// TIA Portal V15.1 export
// export: Created 2024-05-17T05:38:54.2339682Z, ExportSetting WithDefaults, DisplayName Totally Integrated Automation Portal, DisplayVersion V15.1 Update 5, DisplayName TIA Portal Openness, DisplayVersion V15.1 Update 5, DisplayName SINAMICS Startdrive Advanced, DisplayVersion V15.1, DisplayName G130, G150, S120, S150, SINAMICS MV, S210, DisplayVersion V15.1, DisplayName G110M, G120, G120C, G120D, G120P, DisplayVersion V15.1, DisplayName STEP 7 Professional, DisplayVersion V15.1 Update 5, DisplayName STEP 7 Safety, DisplayVersion V15.1, DisplayName WinCC Professional, DisplayVersion V15.1 Update 5, DisplayName SIMATIC Visualization Architect, DisplayVersion V15.1
FUNCTION_BLOCK "LAndonReqVCG"   // FB6050, FBD
TITLE = FB6050: LandonReq / FB6050: LandonReq VCG
{ S7_Optimized_Access := 'FALSE' }
VERSION : 0.1
// =============================================================================
// This module:
//  * Evaluate the Pullcord request to trigger an ANDON event
//  * Gather and organise the data to send to IT shopfloor
//  * Send data to Andon Server on change (buffers only when changed and after 30 
//    sec without an active send)
// =============================================================================
// 08/06/2017: Added Lmaintenancesel
//                       changed Send done to local varible
// 14/02/2017: APPROVAL TEST WITH IT
// 07/12/2106: Expanded StationId to 14 characters
// ============================================================================
// This module:25/11/2016
//  * Evaluate the HCall request to trigger an ANDON event
//  * Gather and organise the data to send to IT shopfloor
//  * Send data to Andon Server on change (buffers only when changed and after 30 
//    sec without an active send)
// ============================================================================
// stored: AutoNumber false, IsIECCheckEnabled false, SetENOAutomatically False, UDAEnableTagReadback false
   VAR_INPUT
      I_WaitingInput { ExternalAccessible := 'False'; ExternalVisible := 'False'; ExternalWritable := 'False'} : Bool;   // I: Not enough bodies on input
      I_WaitingOutput { ExternalAccessible := 'False'; ExternalVisible := 'False'; ExternalWritable := 'False'} : Bool;   // I: Can't deliver body on output
      I_LineStop { ExternalAccessible := 'False'; ExternalVisible := 'False'; ExternalWritable := 'False'} : Bool;   // I: Line Stop
      I_AutoZoneOverCycle { ExternalAccessible := 'False'; ExternalVisible := 'False'; ExternalWritable := 'False'} : Bool;   // I: Automatic unit has exceeded reference time
      I_Operator1OverCycle { ExternalAccessible := 'False'; ExternalVisible := 'False'; ExternalWritable := 'False'} : Bool;   // I: Operator has exceeded reference time
      I_Operator2OverCycle { ExternalAccessible := 'False'; ExternalVisible := 'False'; ExternalWritable := 'False'} : Bool;   // I: Operator has exceeded reference time
      I_Operator3OverCycle { ExternalAccessible := 'False'; ExternalVisible := 'False'; ExternalWritable := 'False'} : Bool;   // I: Operator has exceeded reference time
      I_Operator4OverCycle { ExternalAccessible := 'False'; ExternalVisible := 'False'; ExternalWritable := 'False'} : Bool;   // I: Operator has exceeded reference time
      I_Operator5OverCycle { ExternalAccessible := 'False'; ExternalVisible := 'False'; ExternalWritable := 'False'} : Bool;   // I: Operator has exceeded reference time
      I_Mask { ExternalAccessible := 'False'; ExternalVisible := 'False'; ExternalWritable := 'False'} : Bool;   // I: Mask Andon
   END_VAR
   VAR_IN_OUT
      IO_Modes : "Modes";   // IO: Modes
      IO_VD : "VDComm";   // IO: VDCOM
      IO_AndonStatusVCG : "AndonStatusVCG";   // IO: AndonStatus / IO: AndonStatus <-> Supervision
      IO_AndonDataExchange : "AndonDataExchangeVCG";   // IO: AndonDataExchange
      H_HMI : "H_HMI";   // IO: HMO
      H_AndonReq : "H_AndonReqVCG";   // IO: H_Andon Req
      C_Config : "AndonConfigVCG";   // IO: AndonConfig
   END_VAR
   VAR DB_SPECIFIC
      HCall0 { ExternalAccessible := 'False'; ExternalVisible := 'False'; ExternalWritable := 'False'} : Bool;   // Request andon / Request andon from HMI
      HMI_ReqMuteAndon { ExternalAccessible := 'False'; ExternalVisible := 'False'; ExternalWritable := 'False'} : Bool;   // Mute Andon
      EnableAndonHumanCall { ExternalAccessible := 'False'; ExternalVisible := 'False'; ExternalWritable := 'False'} : Bool := TRUE;   // Bit Used to ENABLE or DISABLE Andon Pullcords BY VAT TABLE FOR DEPLOYMENT ONLY
      SendTriggerFromApp { ExternalAccessible := 'False'; ExternalVisible := 'False'; ExternalWritable := 'False'} : Bool;   // PF used to initiate a message send
      SendRequestFromApp { ExternalAccessible := 'False'; ExternalVisible := 'False'; ExternalWritable := 'False'} : Bool;   // Send Command by application
      ResetNewDataFromApp { ExternalAccessible := 'False'; ExternalVisible := 'False'; ExternalWritable := 'False'} : Bool;   // Trigger by application to reset output "NewData"
      SendBufferValue { ExternalAccessible := 'False'; ExternalVisible := 'False'; ExternalWritable := 'False'} : Bool;   // Send buffer Value
      TempBufferValueHasChanged { ExternalAccessible := 'False'; ExternalVisible := 'False'; ExternalWritable := 'False'} : Bool;   // Buffer value has changed
      TempHCall0Toggle { ExternalAccessible := 'False'; ExternalVisible := 'False'; ExternalWritable := 'False'} : Bool;   // Hcall 0 Toggle
      TempMuteSound { ExternalAccessible := 'False'; ExternalVisible := 'False'; ExternalWritable := 'False'} : Bool;   // Mute Sound
      TempPfMuteSound { ExternalAccessible := 'False'; ExternalVisible := 'False'; ExternalWritable := 'False'} : Bool;   // PF Mute sound
      SendDoneToApp { ExternalAccessible := 'False'; ExternalVisible := 'False'; ExternalWritable := 'False'} : Bool;   // Send Done to App
      NewMessageToApp { ExternalAccessible := 'False'; ExternalVisible := 'False'; ExternalWritable := 'False'} : Bool;   // New Messagge to app
      ResetVDComm { ExternalAccessible := 'False'; ExternalVisible := 'False'; ExternalWritable := 'False'} : Bool;   // Reset VD communication upon timeout
      TempAndonHCallOld { ExternalAccessible := 'False'; ExternalVisible := 'False'; ExternalWritable := 'False'} : DWord;   // i: Andon Hcall Dword previous cycle / Andon Hcall Dword previous cycle
      OldControlDWord2 { ExternalAccessible := 'False'; ExternalVisible := 'False'; ExternalWritable := 'False'} : DWord;   // Save the controlword in the DB
      AndonCtrlDword { ExternalAccessible := 'False'; ExternalVisible := 'False'; ExternalWritable := 'False'} : DWord;   // Temp: Andon status bits control Dword
      AndonCtrlDwordOld { ExternalAccessible := 'False'; ExternalVisible := 'False'; ExternalWritable := 'False'} : DWord;   // Temp: Andon control Dword previous cycle
      OldAndonBuffer1Amount { ExternalAccessible := 'False'; ExternalVisible := 'False'; ExternalWritable := 'False'} : Int;   // Old buffer value
      OldAndonBuffer2Amount { ExternalAccessible := 'False'; ExternalVisible := 'False'; ExternalWritable := 'False'} : Int;   // Old buffer value
      OldAndonBuffer3Amount { ExternalAccessible := 'False'; ExternalVisible := 'False'; ExternalWritable := 'False'} : Int;   // Old buffer value
      OldAndonBuffer4Amount { ExternalAccessible := 'False'; ExternalVisible := 'False'; ExternalWritable := 'False'} : Int;   // Old buffer value
      OldAndonBuffer5Amount { ExternalAccessible := 'False'; ExternalVisible := 'False'; ExternalWritable := 'False'} : Int;   // Old buffer value
      OldAndonBuffer6Amount { ExternalAccessible := 'False'; ExternalVisible := 'False'; ExternalWritable := 'False'} : Int;   // Old buffer value
      OldAndonBuffer7Amount { ExternalAccessible := 'False'; ExternalVisible := 'False'; ExternalWritable := 'False'} : Int;   // Old buffer value
      OldAndonBuffer8Amount { ExternalAccessible := 'False'; ExternalVisible := 'False'; ExternalWritable := 'False'} : Int;   // Old buffer value
      TON_AlarmCFilterTime { ExternalAccessible := 'False'; ExternalVisible := 'False'; ExternalWritable := 'False'} : IEC_TIMER;   // Alarm C filterTime / TON Alarm C filterTime
      TON_SendBufferValue { ExternalAccessible := 'False'; ExternalVisible := 'False'; ExternalWritable := 'False'} : IEC_TIMER;   // TON send buffervalues
   END_VAR
   VAR
      AndonSubSystem { ExternalAccessible := 'False'; ExternalVisible := 'False'; ExternalWritable := 'False'} : "LVDComSubSystemS7-1500";   // Andon Subsystem
   END_VAR
   VAR DB_SPECIFIC
      Edge { ExternalAccessible := 'False'; ExternalVisible := 'False'; ExternalWritable := 'False'} : Array[0..31] of Bool;   // Edges
   END_VAR
   VAR
      LToggle_HCall0 { ExternalAccessible := 'False'; ExternalVisible := 'False'; ExternalWritable := 'False'} : "LToggle";   // Toggle HCall
      LToggle_MuteSound { ExternalAccessible := 'False'; ExternalVisible := 'False'; ExternalWritable := 'False'} : "LToggle";   // Toggle Mutesound
   END_VAR
   VAR DB_SPECIFIC
      SendToVDTimeOut { ExternalAccessible := 'False'; ExternalVisible := 'False'; ExternalWritable := 'False'} : TON_TIME;
      H_CommissioningMode { ExternalAccessible := 'False'; ExternalVisible := 'False'; ExternalWritable := 'False'} : Bool;
      H_TestOPOT1 { ExternalAccessible := 'False'; ExternalVisible := 'False'; ExternalWritable := 'False'} : Bool;   // HMI PB for simulating Operator Overtime 1
      H_TestOPOT2 { ExternalAccessible := 'False'; ExternalVisible := 'False'; ExternalWritable := 'False'} : Bool;   // HMI PB for simulating Operator Overtime 2
      H_TestOPOT3 { ExternalAccessible := 'False'; ExternalVisible := 'False'; ExternalWritable := 'False'} : Bool;   // HMI PB for simulating Operator Overtime 3
      H_TestOPOT4 { ExternalAccessible := 'False'; ExternalVisible := 'False'; ExternalWritable := 'False'} : Bool;   // HMI PB for simulating Operator Overtime 4
      H_TestOPOT5 { ExternalAccessible := 'False'; ExternalVisible := 'False'; ExternalWritable := 'False'} : Bool;   // HMI PB for simulating Operator Overtime 5
      H_TestAutomode { ExternalAccessible := 'False'; ExternalVisible := 'False'; ExternalWritable := 'False'} : Bool;   // HMI PB for simulating Automode ON
      H_TestAlarmC { ExternalAccessible := 'False'; ExternalVisible := 'False'; ExternalWritable := 'False'} : Bool;   // HMI PB for simulating AlarmC ON
      H_TestWaitingInput { ExternalAccessible := 'False'; ExternalVisible := 'False'; ExternalWritable := 'False'} : Bool;   // HMI PB for simulating WaitingInput ON
      H_TestWaitingOutput { ExternalAccessible := 'False'; ExternalVisible := 'False'; ExternalWritable := 'False'} : Bool;   // HMI PB for simulating WaitingOutput ON
      H_TestEQOT { ExternalAccessible := 'False'; ExternalVisible := 'False'; ExternalWritable := 'False'} : Bool;   // HMI PB for simulating Equipment Overtime
      H_TestLineStop { ExternalAccessible := 'False'; ExternalVisible := 'False'; ExternalWritable := 'False'} : Bool;   // HMI PB for simulating LineStop ON
      H_TestManualMode { ExternalAccessible := 'False'; ExternalVisible := 'False'; ExternalWritable := 'False'} : Bool;   // HMI PB for simulating Manualmode ON
      TOF_Mute { ExternalAccessible := 'False'; ExternalVisible := 'False'; ExternalWritable := 'False'} : IEC_TIMER;   // Alarm C filterTime / TON Alarm C filterTime
      MuteSountTOF { ExternalAccessible := 'False'; ExternalVisible := 'False'; ExternalWritable := 'False'} : TOF_TIME;
   END_VAR
   VAR_TEMP   // added for the SCL form of the ladder/FBD networks
      _w1 : Bool;
      _w2 : Bool;
      _w3 : Bool;
   END_VAR
BEGIN

REGION Network 1: **** 1 - Inputs **** HMI Commands
   // Extract The Commands From HMICmd / @@Extract The Commands From HMICmd
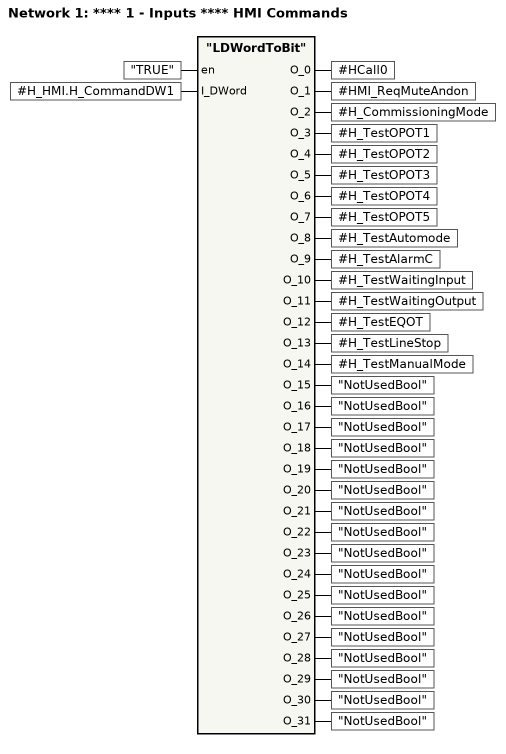
   IF "TRUE" THEN
       "LDWordToBit"(I_DWord := #H_HMI.H_CommandDW1,
                     O_0 => #HCall0,
                     O_1 => #HMI_ReqMuteAndon,
                     O_2 => #H_CommissioningMode,
                     O_3 => #H_TestOPOT1,
                     O_4 => #H_TestOPOT2,
                     O_5 => #H_TestOPOT3,
                     O_6 => #H_TestOPOT4,
                     O_7 => #H_TestOPOT5,
                     O_8 => #H_TestAutomode,
                     O_9 => #H_TestAlarmC,
                     O_10 => #H_TestWaitingInput,
                     O_11 => #H_TestWaitingOutput,
                     O_12 => #H_TestEQOT,
                     O_13 => #H_TestLineStop,
                     O_14 => #H_TestManualMode,
                     O_15 => "NotUsedBool",
                     O_16 => "NotUsedBool",
                     O_17 => "NotUsedBool",
                     O_18 => "NotUsedBool",
                     O_19 => "NotUsedBool",
                     O_20 => "NotUsedBool",
                     O_21 => "NotUsedBool",
                     O_22 => "NotUsedBool",
                     O_23 => "NotUsedBool",
                     O_24 => "NotUsedBool",
                     O_25 => "NotUsedBool",
                     O_26 => "NotUsedBool",
                     O_27 => "NotUsedBool",
                     O_28 => "NotUsedBool",
                     O_29 => "NotUsedBool",
                     O_30 => "NotUsedBool",
                     O_31 => "NotUsedBool");
   END_IF;
END_REGION

REGION Network 2: **** 1 - Inputs **** Combine Controlbits to DWord
   // Bit 0.0 automode (AUTO)
   // Bit 0.1 Operator Requested with 30 second filtertime (OPER)
   // Bit 0.2 Waiting Input (WIP)
   // Bit 0.3 Waiting Output (WOP)
   // Bit 0.4 Operator Overtime (OPOT)
   // Bit 0.5 EquipmentOvertime (EQOT)
   // Bit 0.6 LineStop(LS)
   // Bit 0.7 Mask (MASK)
   // Bit 1.0 Mute Sound by button on station or external function(MUTS)
   // Bit 1.1 Request Teamleader: Request a teamleader when button is pressed on AM0
   //             station or when operator overtime is detetected
   // Bit 1.2 Request ModeZone: when button is pressed on station or when operator  (REQMZ)
   // Bit 1.3 Request Maintenance: when button is pressed on station or when equipment
   // overtime is detetected
   // Bit 1.4 HumanCall (AM0)
   // Bit 1.5 Spare
   // Bit 1.6 Spare
   // Bit 2.0 2.7 spare
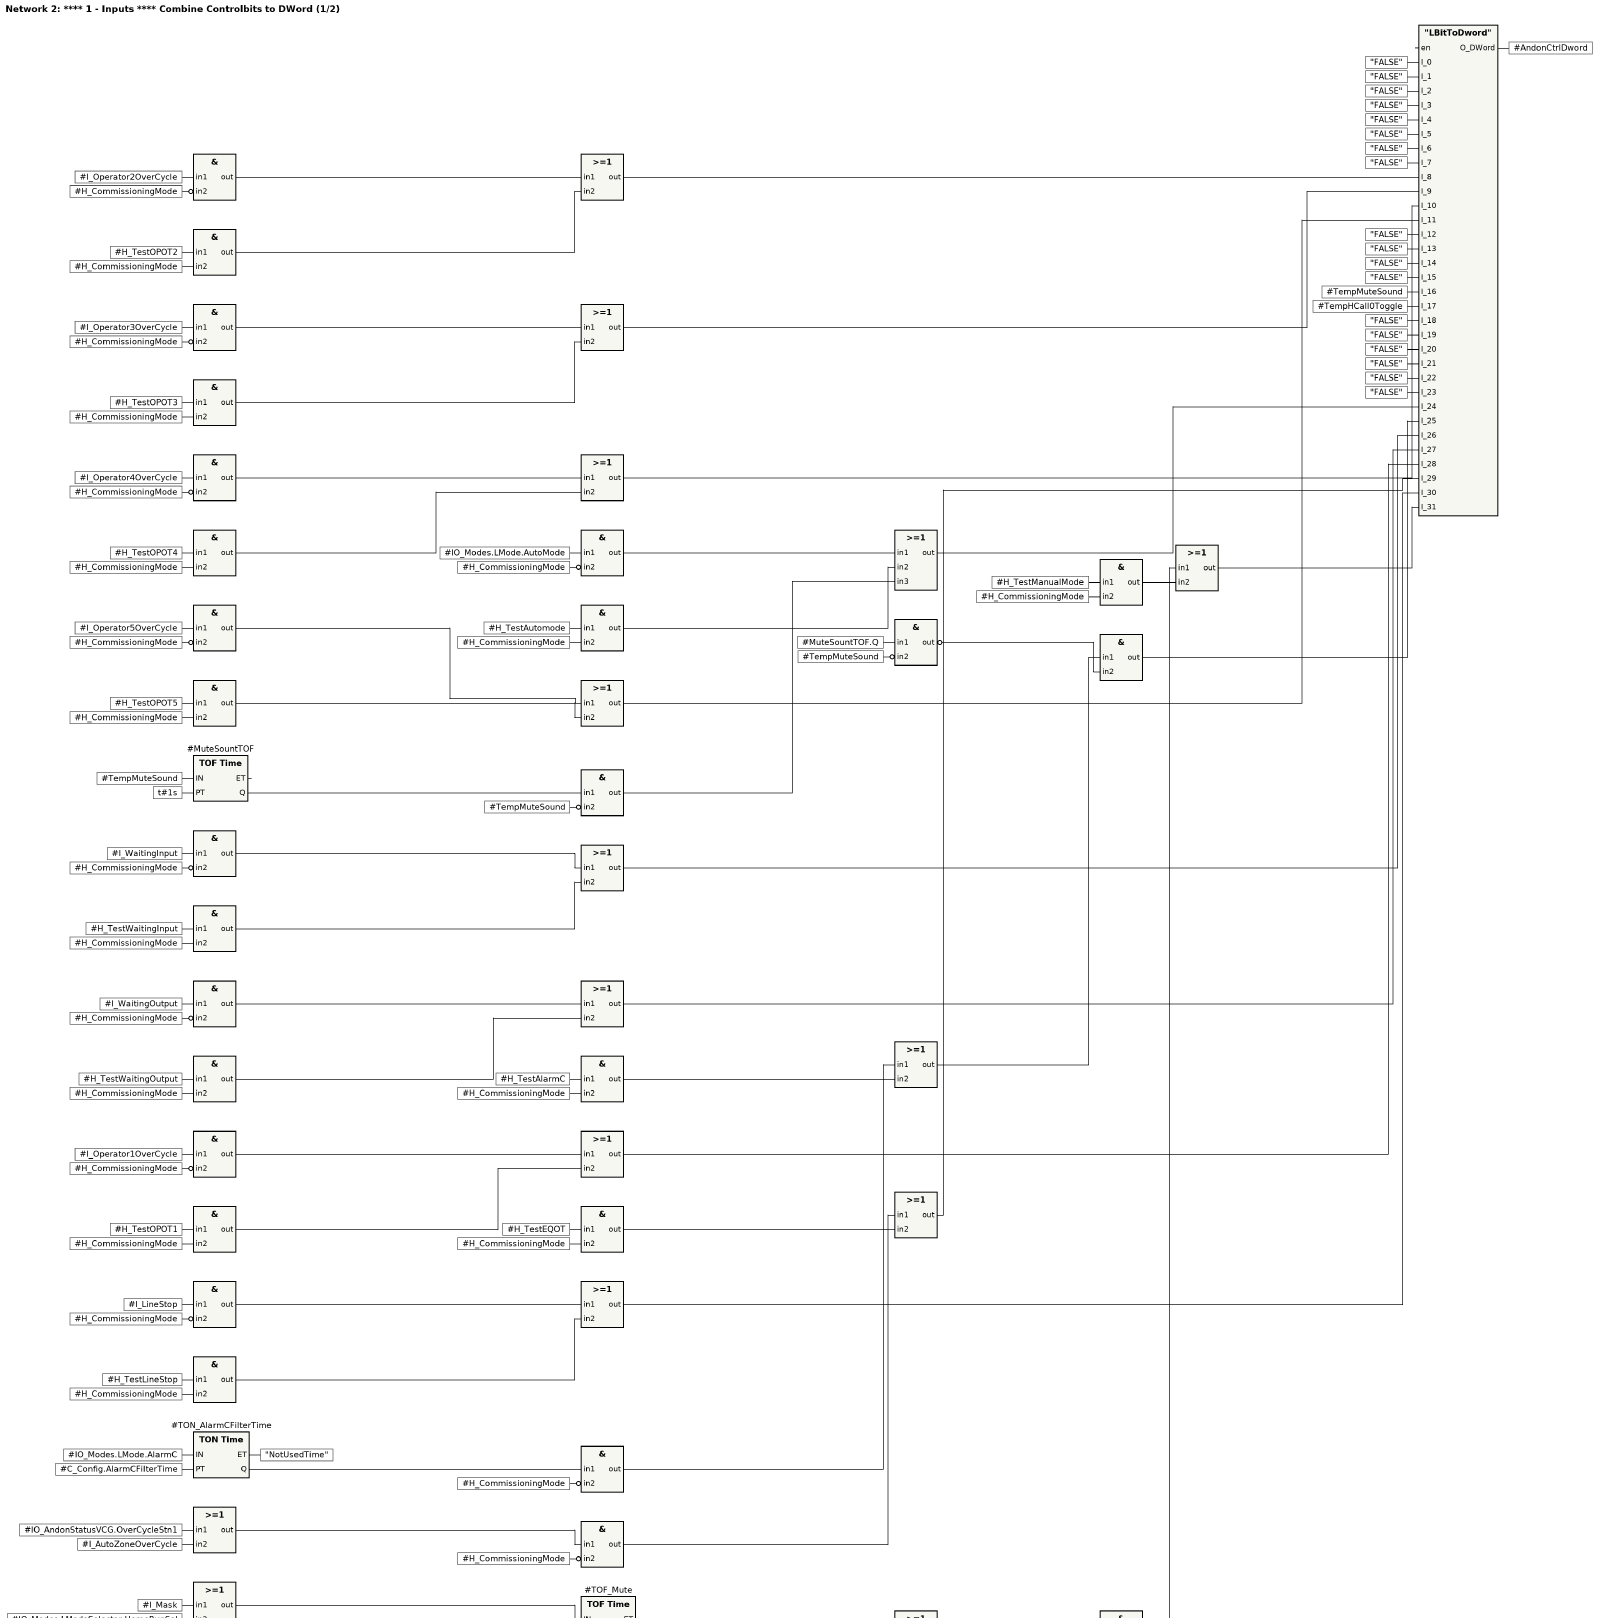
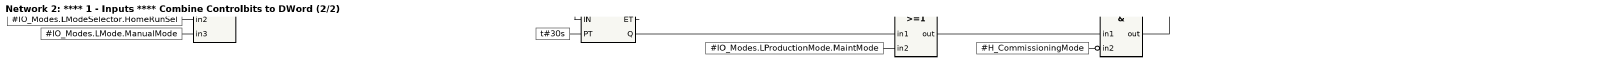
   #MuteSountTOF(IN := #TempMuteSound, PT := t#1s);   // TOF
   #TON_AlarmCFilterTime.TON(IN := #IO_Modes.LMode.AlarmC,
                           PT := #C_Config.AlarmCFilterTime,
                           ET => "NotUsedTime");
   #TOF_Mute.TOF(IN := #I_Mask OR #IO_Modes.LModeSelector.HomeRunSel OR #IO_Modes.LMode.ManualMode, PT := t#30s);
   "LBitToDword"(I_0 := "FALSE",
                 I_1 := "FALSE",
                 I_2 := "FALSE",
                 I_3 := "FALSE",
                 I_4 := "FALSE",
                 I_5 := "FALSE",
                 I_6 := "FALSE",
                 I_7 := "FALSE",
                 I_8 := (#I_Operator2OverCycle AND NOT #H_CommissioningMode) OR (#H_TestOPOT2 AND #H_CommissioningMode),
                 I_9 := (#I_Operator3OverCycle AND NOT #H_CommissioningMode) OR (#H_TestOPOT3 AND #H_CommissioningMode),
                 I_10 := (#I_Operator4OverCycle AND NOT #H_CommissioningMode) OR (#H_TestOPOT4 AND #H_CommissioningMode),
                 I_11 := (#I_Operator5OverCycle AND NOT #H_CommissioningMode) OR (#H_TestOPOT5 AND #H_CommissioningMode),
                 I_12 := "FALSE",
                 I_13 := "FALSE",
                 I_14 := "FALSE",
                 I_15 := "FALSE",
                 I_16 := #TempMuteSound,
                 I_17 := #TempHCall0Toggle,
                 I_18 := "FALSE",
                 I_19 := "FALSE",
                 I_20 := "FALSE",
                 I_21 := "FALSE",
                 I_22 := "FALSE",
                 I_23 := "FALSE",
                 I_24 := (#IO_Modes.LMode.AutoMode AND NOT #H_CommissioningMode) OR (#H_TestAutomode AND #H_CommissioningMode) OR (#MuteSountTOF.Q AND NOT #TempMuteSound),
                 I_25 := ((#TON_AlarmCFilterTime.Q AND NOT #H_CommissioningMode) OR (#H_TestAlarmC AND #H_CommissioningMode)) AND NOT (#MuteSountTOF.Q AND NOT #TempMuteSound),
                 I_26 := (#I_WaitingInput AND NOT #H_CommissioningMode) OR (#H_TestWaitingInput AND #H_CommissioningMode),
                 I_27 := (#I_WaitingOutput AND NOT #H_CommissioningMode) OR (#H_TestWaitingOutput AND #H_CommissioningMode),
                 I_28 := (#I_Operator1OverCycle AND NOT #H_CommissioningMode) OR (#H_TestOPOT1 AND #H_CommissioningMode),
                 I_29 := ((#IO_AndonStatusVCG.OverCycleStn1 OR #I_AutoZoneOverCycle) AND NOT #H_CommissioningMode) OR (#H_TestEQOT AND #H_CommissioningMode),
                 I_30 := (#I_LineStop AND NOT #H_CommissioningMode) OR (#H_TestLineStop AND #H_CommissioningMode),
                 I_31 := ((#TOF_Mute.Q OR #IO_Modes.LProductionMode.MaintMode) AND NOT #H_CommissioningMode) OR (#H_TestManualMode AND #H_CommissioningMode),
                 O_DWord => #AndonCtrlDword);
END_REGION

REGION Network 3: **** - Communication ***** VDCom Subsystem (NEEDS CHECKING) / **** 3.1 - Communication ***** VDCom Subsystem
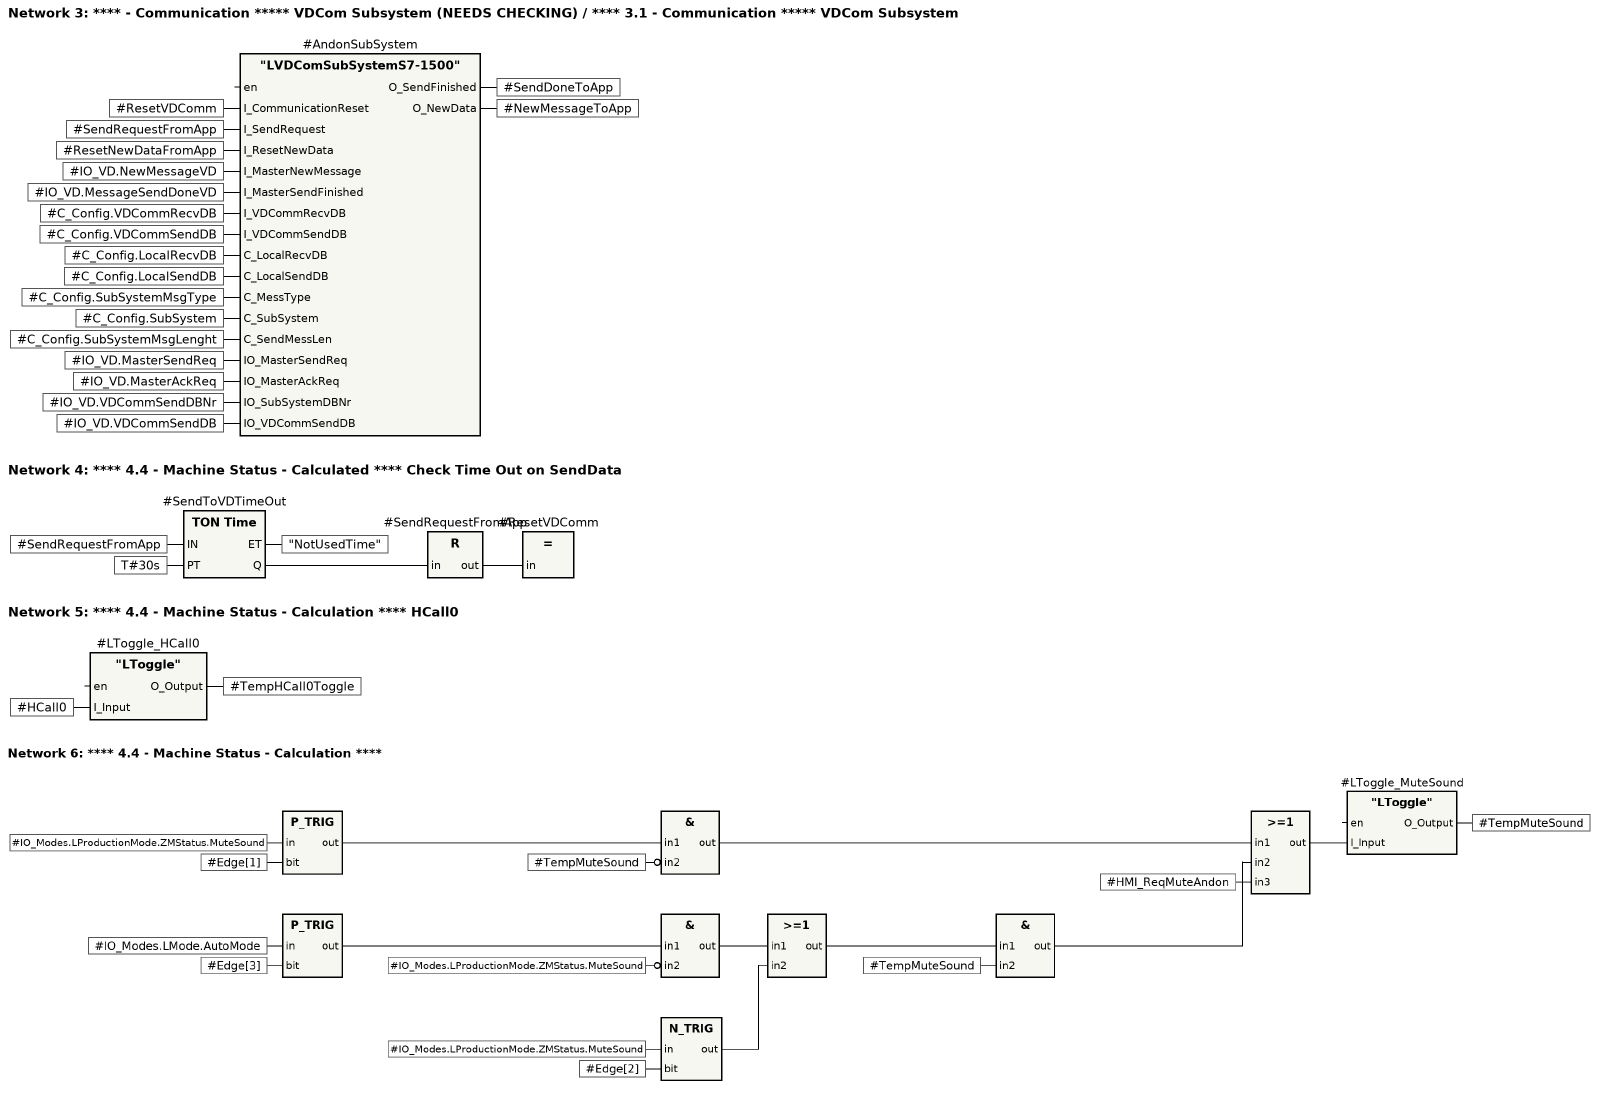
   #AndonSubSystem(I_CommunicationReset := #ResetVDComm,   // "LVDComSubSystemS7-1500"
                   I_SendRequest := #SendRequestFromApp,
                   I_ResetNewData := #ResetNewDataFromApp,
                   I_MasterNewMessage := #IO_VD.NewMessageVD,
                   I_MasterSendFinished := #IO_VD.MessageSendDoneVD,
                   I_VDCommRecvDB := #C_Config.VDCommRecvDB,
                   I_VDCommSendDB := #C_Config.VDCommSendDB,
                   C_LocalRecvDB := #C_Config.LocalRecvDB,
                   C_LocalSendDB := #C_Config.LocalSendDB,
                   C_MessType := #C_Config.SubSystemMsgType,
                   C_SubSystem := #C_Config.SubSystem,
                   C_SendMessLen := #C_Config.SubSystemMsgLenght,
                   IO_MasterSendReq := #IO_VD.MasterSendReq,
                   IO_MasterAckReq := #IO_VD.MasterAckReq,
                   IO_SubSystemDBNr := #IO_VD.VDCommSendDBNr,
                   IO_VDCommSendDB := #IO_VD.VDCommSendDB,
                   O_SendFinished => #SendDoneToApp,
                   O_NewData => #NewMessageToApp);
END_REGION

REGION Network 4: **** 4.4 - Machine Status - Calculated **** Check Time Out on SendData
   // Reset Send request when time out elapses
   // Reset the VD communication
   #SendToVDTimeOut(IN := #SendRequestFromApp, PT := T#30s, ET => "NotUsedTime");   // TON
   IF #SendToVDTimeOut.Q THEN #SendRequestFromApp := FALSE; END_IF;
   #ResetVDComm := #SendToVDTimeOut.Q;
END_REGION

REGION Network 5: **** 4.4 - Machine Status - Calculation **** HCall0
   // Toggle function for HCall
   #LToggle_HCall0(I_Input := #HCall0, O_Output => #TempHCall0Toggle);   // "LToggle"
END_REGION

REGION Network 6: **** 4.4 - Machine Status - Calculation ****
   #_w1 := #IO_Modes.LProductionMode.ZMStatus.MuteSound AND NOT #Edge[1];   // rising edge
   #Edge[1] := #IO_Modes.LProductionMode.ZMStatus.MuteSound;
   #_w2 := #IO_Modes.LMode.AutoMode AND NOT #Edge[3];   // rising edge
   #Edge[3] := #IO_Modes.LMode.AutoMode;
   #_w3 := NOT #IO_Modes.LProductionMode.ZMStatus.MuteSound AND #Edge[2];   // falling edge
   #Edge[2] := #IO_Modes.LProductionMode.ZMStatus.MuteSound;
   #LToggle_MuteSound(I_Input := (#_w1 AND NOT #TempMuteSound) OR (((#_w2 AND NOT #IO_Modes.LProductionMode.ZMStatus.MuteSound) OR #_w3) AND #TempMuteSound) OR #HMI_ReqMuteAndon,   // "LToggle"
                      O_Output => #TempMuteSound);
END_REGION

REGION Network 7: **** 4.4 - Machine Status - Calculation **** SEND BUFFERS
   // Determine if a buffervalue has changed (Values are only copied to "old" Value 
   // when a send is active
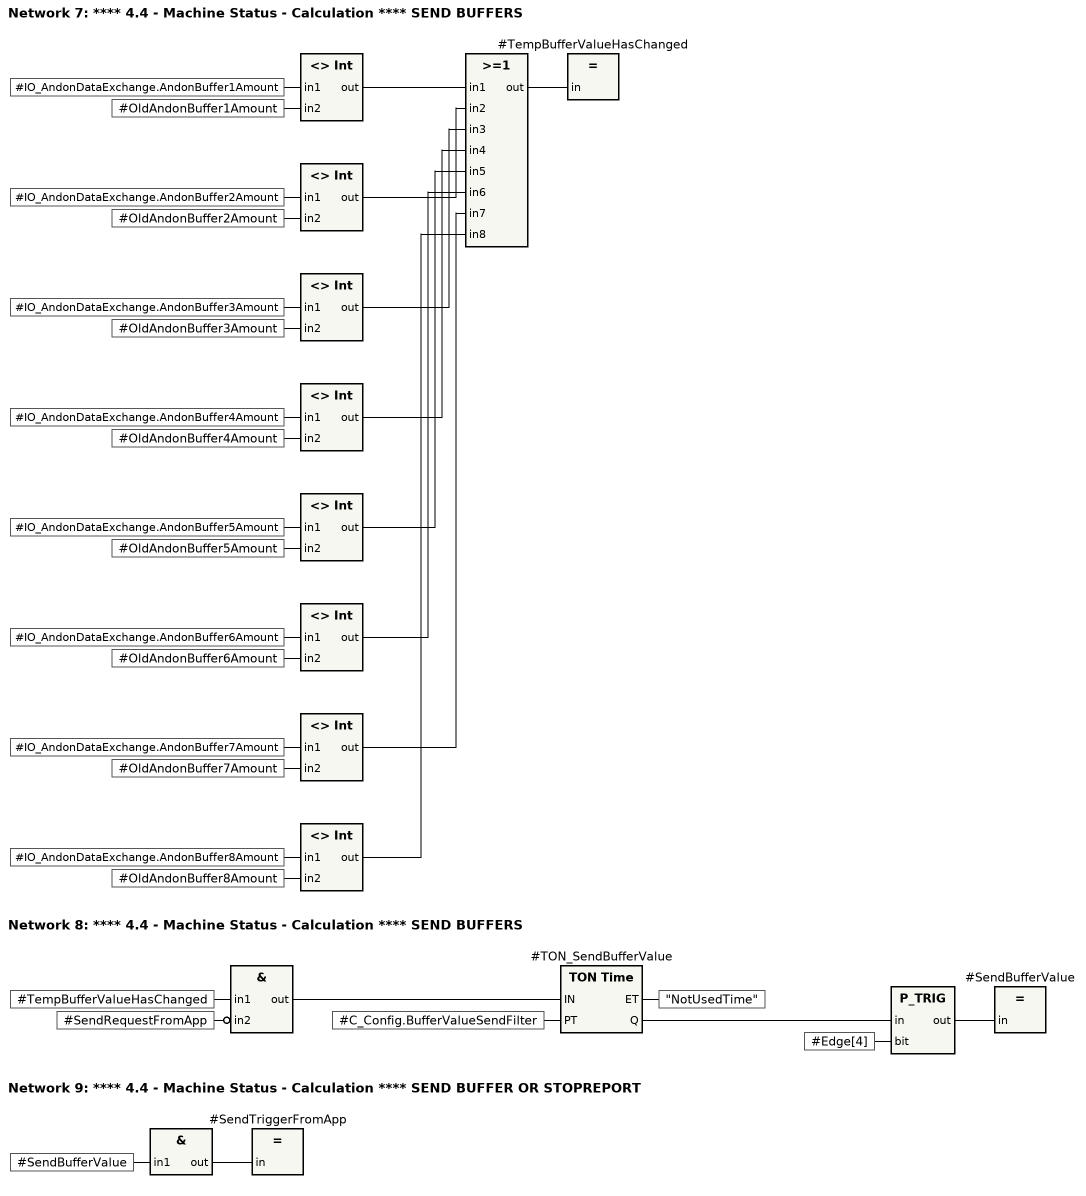
   #TempBufferValueHasChanged := (#IO_AndonDataExchange.AndonBuffer1Amount <> #OldAndonBuffer1Amount) OR (#IO_AndonDataExchange.AndonBuffer2Amount <> #OldAndonBuffer2Amount) OR (#IO_AndonDataExchange.AndonBuffer3Amount <> #OldAndonBuffer3Amount) OR (#IO_AndonDataExchange.AndonBuffer4Amount <> #OldAndonBuffer4Amount) OR (#IO_AndonDataExchange.AndonBuffer5Amount <> #OldAndonBuffer5Amount) OR (#IO_AndonDataExchange.AndonBuffer6Amount <> #OldAndonBuffer6Amount) OR (#IO_AndonDataExchange.AndonBuffer7Amount <> #OldAndonBuffer7Amount) OR (#IO_AndonDataExchange.AndonBuffer8Amount <> #OldAndonBuffer8Amount);
END_REGION

REGION Network 8: **** 4.4 - Machine Status - Calculation **** SEND BUFFERS
   // Send buffer value to VD when last message was 60 seconds ago but do not send 
   // when sending is in progress
   #TON_SendBufferValue.TON(IN := #TempBufferValueHasChanged AND NOT #SendRequestFromApp,
                           PT := #C_Config.BufferValueSendFilter,
                           ET => "NotUsedTime");
   #_w1 := #TON_SendBufferValue.Q AND NOT #Edge[4];   // rising edge
   #Edge[4] := #TON_SendBufferValue.Q;
   #SendBufferValue := #_w1;
END_REGION

REGION Network 9: **** 4.4 - Machine Status - Calculation **** SEND BUFFER OR STOPREPORT
   #SendTriggerFromApp := #SendBufferValue;
END_REGION

NETWORK
TITLE = **** 4.6 - Machine status - Indication **** OPEN CONFIGURATION
// Open the DB used for sending data to ANDON VDCOM
      OPN   #C_Config.LocalSendDB;

NETWORK
TITLE = **** 4.6 - Machine status - Indication **** PREPARE MESSAGE HEADER SHOP ID
// TRANSFER THE SHOP ID INTO THE SEND DB
      L     #C_Config.ShopID[1];
      T     %DBB10;
      L     #C_Config.ShopID[2];
      T     %DBB11;
      L     #C_Config.ShopID[3];
      T     %DBB12;


NETWORK
TITLE = **** 4.6 - Machine status - Indication **** PREPARE MESSAGE HEADER STATION ID
      L     #C_Config.StationID[1];
      T     %DBB13;
      L     #C_Config.StationID[2];
      T     %DBB14;
      L     #C_Config.StationID[3];
      T     %DBB15;
      L     #C_Config.StationID[4];
      T     %DBB16;
      L     #C_Config.StationID[5];
      T     %DBB17;
      L     #C_Config.StationID[6];
      T     %DBB18;
      L     #C_Config.StationID[7];
      T     %DBB19;
      L     #C_Config.StationID[8];
      T     %DBB20;
      L     #C_Config.StationID[9];
      T     %DBB21;
      L     #C_Config.StationID[10];
      T     %DBB22;
      L     #C_Config.StationID[11];
      T     %DBB23;
      L     #C_Config.StationID[12];
      T     %DBB24;
      L     #C_Config.StationID[13];
      T     %DBB25;
      L     #C_Config.StationID[14];
      T     %DBB26;


NETWORK
TITLE = **** 4.6 - Machine status - Indication **** PREPARE MESSAGE BODY
// COPY CONTROL DW TO SEND DB
      L     #AndonCtrlDword;
      T     %DBD28;

NETWORK
TITLE = **** 4.6 - Machine status - Indication **** PREPARE MESSAGE BODY
// COPY CONTROL WORD TO SEND DB
      L     #IO_AndonDataExchange.AndonHCallActive;
      T     %DBD32;

NETWORK
TITLE = **** 4.6 - Machine status - Indication **** PREPARE MESSAGE BODY
// TRANSFER BUFFER VALUES TO SEND DB
// TRANSFER VALUES BUFFER 1
      L     #IO_AndonDataExchange.AndonBuffer1Amount;
      T     %DBW36;
      L     #IO_AndonDataExchange.AndonBuffer1Maximum;
      T     %DBW38;
// TRANSFER VALUES BUFFER 2
      L     #IO_AndonDataExchange.AndonBuffer2Amount;
      T     %DBW40;
      L     #IO_AndonDataExchange.AndonBuffer2Maximum;
      T     %DBW42;
// TRANSFER VALUES BUFFER 3
      L     #IO_AndonDataExchange.AndonBuffer3Amount;
      T     %DBW44;
      L     #IO_AndonDataExchange.AndonBuffer3Maximum;
      T     %DBW46;
// TRANSFER VALUES BUFFER 4
      L     #IO_AndonDataExchange.AndonBuffer4Amount;
      T     %DBW48;
      L     #IO_AndonDataExchange.AndonBuffer4Maximum;
      T     %DBW50;
// TRANSFER VALUES BUFFER 5
      L     #IO_AndonDataExchange.AndonBuffer5Amount;
      T     %DBW52;
      L     #IO_AndonDataExchange.AndonBuffer5Maximum;
      T     %DBW54;
// TRANSFER VALUES BUFFER 6
      L     #IO_AndonDataExchange.AndonBuffer6Amount;
      T     %DBW56;
      L     #IO_AndonDataExchange.AndonBuffer6Maximum;
      T     %DBW58;
// TRANSFER VALUES BUFFER 7
      L     #IO_AndonDataExchange.AndonBuffer7Amount;
      T     %DBW60;
      L     #IO_AndonDataExchange.AndonBuffer7Maximum;
      T     %DBW62;
// TRANSFER VALUES BUFFER 8
      L     #IO_AndonDataExchange.AndonBuffer8Amount;
      T     %DBW64;
      L     #IO_AndonDataExchange.AndonBuffer8Maximum;
      T     %DBW66;

NETWORK
TITLE = **** 4.6 - Machine status - Indication **** SEND MESSAGE BIT
// FIRST 8 Bytes are reserved.
// Compare the first 8 Bytes (64 bits) of the local stack with a precious cycle 
// version
// If there is a difference then execute the SEND: Command
// Before exiting FB Save Current Controlwords to #OldControlDword
// RESET REQUEST TO MASTER WHEN ACK IS RECIEVED
      A     #SendDoneToApp;
      R     #SendRequestFromApp;
      JC    END;

// IF SEND IS BUSY DONT DO ANYTHING
      A     #SendRequestFromApp;
      JC    FINA;

// SEND BUFFER VALUES EVERY 60 SECONDS (TO REDUCE TRAFFIC)
      A     #SendTriggerFromApp;
      JC    SEND;


// COMPARE CONTROL DOUBLE WORD 1
      L     #AndonCtrlDword;  // LOAD ControldWord 1
      L     #AndonCtrlDwordOld;  // LOAD old ControldWord1
      <>D;  // WHEN different Send to VD
      JC    SEND;

//COMPARE CONTROL WORD 2 (WE ONLY WANT TO SEND ONCE SO USE STATION OUT)
      L     #IO_AndonDataExchange.AndonHCallActive;  // LOAD ControlWord 2(with HCalls)
      L     #TempAndonHCallOld;  // LOAD old ControlWord 2

      <>D;  // WHEN different Send to VD
      JC    SEND;

//IF NOTHING CHANGES JUMP TO END
      JU    END;

// SEND TELEGRAM TO IT SHOPFLOOR
SEND: NOP   0;

      S     #SendRequestFromApp;

// ONLY COPY BUFFER VALUES WHEN #SendRequestFromApp IS HIGH

      L     #IO_AndonDataExchange.AndonBuffer1Amount;
      T     #OldAndonBuffer1Amount;
      L     #IO_AndonDataExchange.AndonBuffer2Amount;
      T     #OldAndonBuffer2Amount;
      L     #IO_AndonDataExchange.AndonBuffer3Amount;
      T     #OldAndonBuffer3Amount;
      L     #IO_AndonDataExchange.AndonBuffer4Amount;
      T     #OldAndonBuffer4Amount;
      L     #IO_AndonDataExchange.AndonBuffer5Amount;
      T     #OldAndonBuffer5Amount;
      L     #IO_AndonDataExchange.AndonBuffer6Amount;
      T     #OldAndonBuffer6Amount;
      L     #IO_AndonDataExchange.AndonBuffer7Amount;
      T     #OldAndonBuffer7Amount;
      L     #IO_AndonDataExchange.AndonBuffer8Amount;
      T     #OldAndonBuffer8Amount;

END:  NOP   0;

// COPY VALUES INTO DB
// TRANSFER VALUES TO CONTROLWORD 1
      L     #AndonCtrlDword;  // LOAD ControlWord 1
      T     #AndonCtrlDwordOld;  // TRANSFER to old ControlWord1

// TRANSFER VALUES TO CONTROLWORD 2 TempAndonHCallOld
      L     #IO_AndonDataExchange.AndonHCallActive;
      T     #TempAndonHCallOld;  // Transfer To old ControlWord2

// TRANSFER VALUES TO CONTROLWORD 3


// TRANSFER VALUES TO CONTROLWORD 4



FINA: NOP   0;

REGION Network 17: **** 4.6 - Machine Status - Indication **** Icon Animation / **** 4.6 - Machine Status - Indication **** ICON ANIMATION
   // Icon Animation
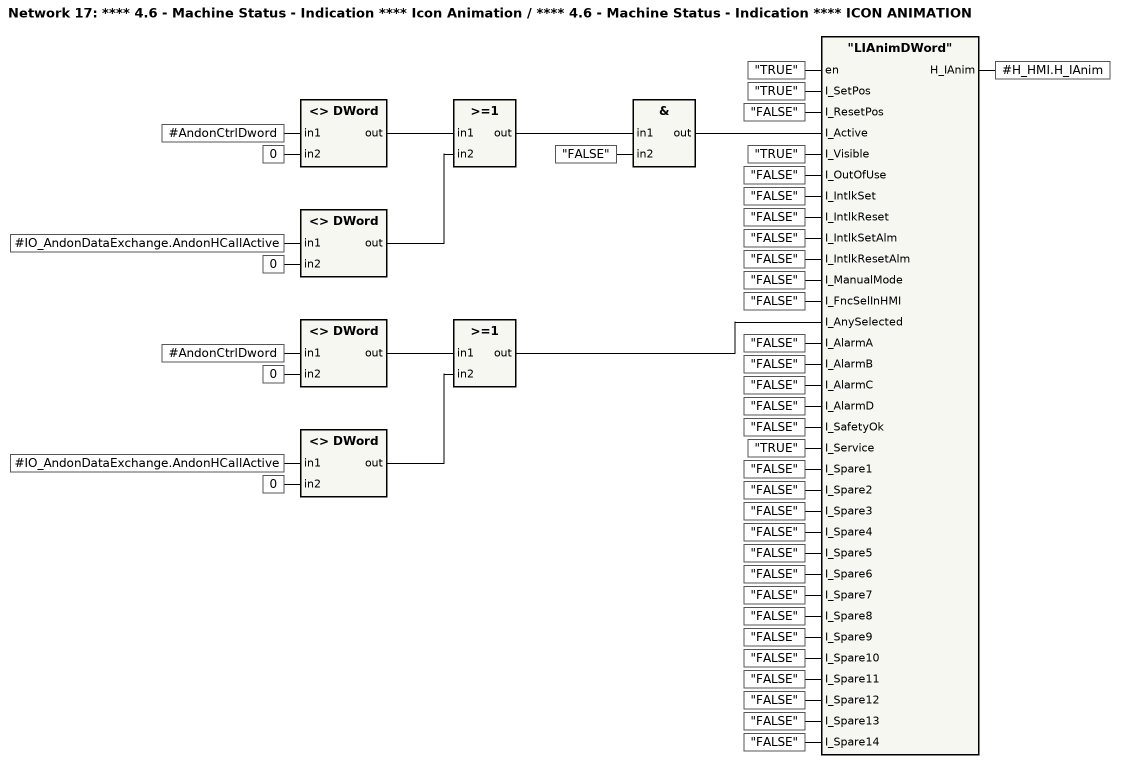
   IF "TRUE" THEN
       "LIAnimDWord"(I_SetPos := "TRUE",
                     I_ResetPos := "FALSE",
                     I_Active := ((#AndonCtrlDword <> 0) OR (#IO_AndonDataExchange.AndonHCallActive <> 0)) AND "FALSE",
                     I_Visible := "TRUE",
                     I_OutOfUse := "FALSE",
                     I_IntlkSet := "FALSE",
                     I_IntlkReset := "FALSE",
                     I_IntlkSetAlm := "FALSE",
                     I_IntlkResetAlm := "FALSE",
                     I_ManualMode := "FALSE",
                     I_FncSelInHMI := "FALSE",
                     I_AnySelected := (#AndonCtrlDword <> 0) OR (#IO_AndonDataExchange.AndonHCallActive <> 0),
                     I_AlarmA := "FALSE",
                     I_AlarmB := "FALSE",
                     I_AlarmC := "FALSE",
                     I_AlarmD := "FALSE",
                     I_SafetyOk := "FALSE",
                     I_Service := "TRUE",
                     I_Spare1 := "FALSE",
                     I_Spare2 := "FALSE",
                     I_Spare3 := "FALSE",
                     I_Spare4 := "FALSE",
                     I_Spare5 := "FALSE",
                     I_Spare6 := "FALSE",
                     I_Spare7 := "FALSE",
                     I_Spare8 := "FALSE",
                     I_Spare9 := "FALSE",
                     I_Spare10 := "FALSE",
                     I_Spare11 := "FALSE",
                     I_Spare12 := "FALSE",
                     I_Spare13 := "FALSE",
                     I_Spare14 := "FALSE",
                     H_IAnim => #H_HMI.H_IAnim);
   END_IF;
END_REGION

REGION Network 18: **** 4.6 - Machine Status - Indication **** Animation / **** 4.6 - Machine Status - Indication **** ANIMATION
   // Animation
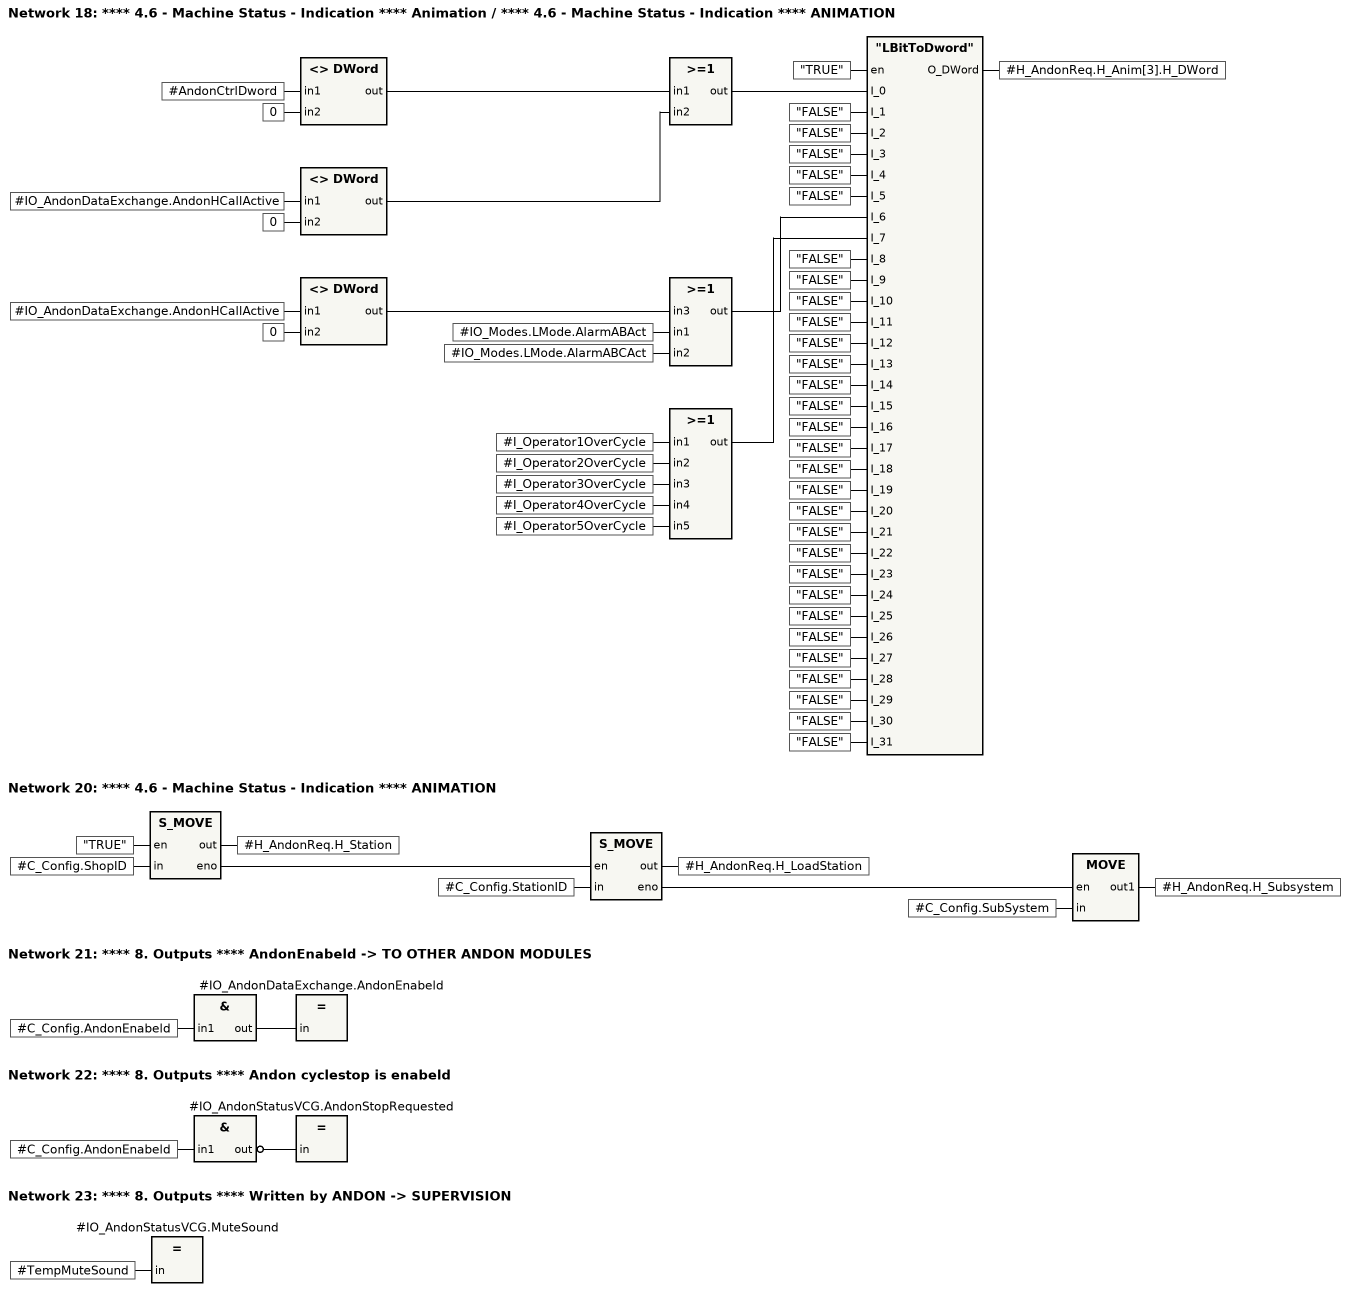
   IF "TRUE" THEN
       "LBitToDword"(I_0 := (#AndonCtrlDword <> 0) OR (#IO_AndonDataExchange.AndonHCallActive <> 0),
                     I_1 := "FALSE",
                     I_2 := "FALSE",
                     I_3 := "FALSE",
                     I_4 := "FALSE",
                     I_5 := "FALSE",
                     I_6 := (#IO_AndonDataExchange.AndonHCallActive <> 0) OR #IO_Modes.LMode.AlarmABAct OR #IO_Modes.LMode.AlarmABCAct,
                     I_7 := #I_Operator1OverCycle OR #I_Operator2OverCycle OR #I_Operator3OverCycle OR #I_Operator4OverCycle OR #I_Operator5OverCycle,
                     I_8 := "FALSE",
                     I_9 := "FALSE",
                     I_10 := "FALSE",
                     I_11 := "FALSE",
                     I_12 := "FALSE",
                     I_13 := "FALSE",
                     I_14 := "FALSE",
                     I_15 := "FALSE",
                     I_16 := "FALSE",
                     I_17 := "FALSE",
                     I_18 := "FALSE",
                     I_19 := "FALSE",
                     I_20 := "FALSE",
                     I_21 := "FALSE",
                     I_22 := "FALSE",
                     I_23 := "FALSE",
                     I_24 := "FALSE",
                     I_25 := "FALSE",
                     I_26 := "FALSE",
                     I_27 := "FALSE",
                     I_28 := "FALSE",
                     I_29 := "FALSE",
                     I_30 := "FALSE",
                     I_31 := "FALSE",
                     O_DWord => #H_AndonReq.H_Anim[3].H_DWord);
   END_IF;
END_REGION

NETWORK
TITLE = **** 4.6 - Machine Status - Indication **** Animation / **** 4.6 - Machine Status - Indication **** ANIMATION
// Visualisation of the controlword
      L     #AndonCtrlDword;
      T     #H_AndonReq.H_Anim[1].H_DWord;
      L     #IO_AndonDataExchange.AndonHCallActive;
      T     #H_AndonReq.H_Anim[2].H_DWord;

REGION Network 20: **** 4.6 - Machine Status - Indication **** ANIMATION
   // Visualisation of the ShopID and the StationID
   IF "TRUE" THEN
       #H_AndonReq.H_Station := #C_Config.ShopID;
       #H_AndonReq.H_LoadStation := #C_Config.StationID;
       #H_AndonReq.H_Subsystem := #C_Config.SubSystem;
   END_IF;
END_REGION

REGION Network 21: **** 8. Outputs **** AndonEnabeld -> TO OTHER ANDON MODULES
   #IO_AndonDataExchange.AndonEnabeld := #C_Config.AndonEnabeld;
END_REGION

REGION Network 22: **** 8. Outputs **** Andon cyclestop is enabeld
   #IO_AndonStatusVCG.AndonStopRequested := NOT #C_Config.AndonEnabeld;
END_REGION

REGION Network 23: **** 8. Outputs **** Written by ANDON -> SUPERVISION
   #IO_AndonStatusVCG.MuteSound := #TempMuteSound;
END_REGION

REGION Network 24: **** 8. Outputs **** Written by ANDON -> SUPERVISION
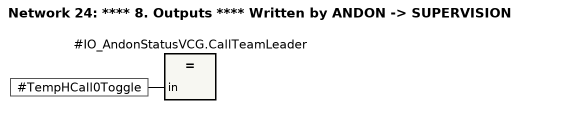
   #IO_AndonStatusVCG.CallTeamLeader := #TempHCall0Toggle;
END_REGION
END_FUNCTION_BLOCK
